{attribute 'qualified_only'}
{attribute 'to_string'}
TYPE E_ProtoWireType :
(
	Varint          := 0,
	Fixed64         := 1,
	LengthDelimited := 2,
	Fixed32         := 5
);
END_TYPE

(* stored: Version 1.1.0.1
   DUT E_ProtoWireType: Id {eda460e0-5e7e-4c57-a7ae-0ce12aae9687} *)
